INTERFACE I_Argument

METHOD PUBLIC M_AddBOOL : I_Argument
VAR_INPUT
	nValue:				LINT;
END_VAR
END_METHOD

METHOD PUBLIC M_AddINT : I_Argument
VAR_INPUT
	nValue:				LINT;
END_VAR
END_METHOD

METHOD PUBLIC M_AddREAL : I_Argument
VAR_INPUT
	fValue:				LREAL;
	nDecimals:			USINT;
END_VAR
END_METHOD

METHOD PUBLIC M_AddSTRING : I_Argument
VAR_INPUT
	sValue:				STRING(255);
END_VAR
END_METHOD

METHOD PUBLIC M_AddTIME : I_Argument
VAR_INPUT
	tValue:				TIME;
END_VAR
END_METHOD

METHOD PUBLIC M_Clear : I_Argument
VAR_INPUT
END_VAR
END_METHOD

PROPERTY PUBLIC P_Value : string(255)
GET
END_GET
END_PROPERTY

END_INTERFACE

(* stored: Version 1.1.0.1
   Itf I_Argument: Id {6070f7e3-601d-44ff-953b-e02d5e046b3f}
   Method M_AddBOOL: Id {4a4232c5-0b26-4f8c-ad4a-57193de9aa82}
   Method M_AddINT: Id {99a67206-55c1-420d-bfe5-b508362e690a}
   Method M_AddREAL: Id {1ad60c9b-cb74-4a8f-bb0e-612d270c055f}
   Method M_AddSTRING: Id {414031c3-c7b6-4eea-9f37-5e0792bcf60a}
   Method M_AddTIME: Id {71f3c0ef-d656-473b-a742-2f0eba5b6965}
   Method M_Clear: Id {6ae742a7-b2b9-4d22-b51b-9a085a158100}
   Property P_Value: Id {0503188b-97cc-41df-8f7e-52f232810f0c}
   Get Get: Id {c58f5a69-aa2b-4993-9224-a484f99c2b8e} *)
